GLOBALCONSTANTS PKP_2200 (* Global constants *)
  (* Standard: 61499-1; Description: Copyright (c) 2023 HR Agrartechnik GmbH This program and the accompanying materials are made available under the terms of the Eclipse Public License 2.0 which is available at https://www.eclipse.org/legal/epl-2.0/ SPDX-License-Identifier: EPL-2.0 *)
  (* Version 1.0, 2023-10-22, Franz Höpfinger, HR Agrartechnik GmbH *)
  PACKAGE BlinkMarine::io::DI;
  IMPORT eclipse4diac::core::TypeHash;
  VAR_GLOBAL CONSTANT
    PKP_2200_DEFAULT : USINT := USINT#16#21;
  END_VAR
END_GLOBALCONSTANTS
